{attribute 'GeneratedUsingTerminal: AT2050-0500-0016'}
{attribute addProperty BoxType "AT2050-0500-0016"}
{attribute addProperty Id "A_0097_AT2025_5250_0018_AT2025_5250AT2025_33A3DF1B80"}
{attribute addProperty CRC "329198353"}
{attribute addProperty Size "80"}
TYPE A_0047_AT2050_0500_0016_139F2B11 EXTENDS AT2050_2EA6C9BF :
STRUCT
	{attribute addProperty Name "A_0097_AT2025_5250_0018_AT2025_5250"}
	{attribute addProperty PreviousPort "A_0047(AT2050-0500-0016) : B"}
	A_0097_AT2025_5250_0018_AT2025_5250 : AT2025_33A3DF1B;
END_STRUCT
END_TYPE

(* stored: Version 1.2.0.0, ProductVersion 3.1.4024.9
   DUT A_0047_AT2050_0500_0016_139F2B11: Id {92b52b8a-7a70-46d4-97be-b542efb62a04} *)
